(* IEC 61131-3 sources: wago_2pump_ebm_fans/PFC200_G2_2ETH_RS_CAN_DPS_T.device.xml.v3^/Plc Logic.plclogic.xml.v3^/Application.application.xml.v3^, 5 files *)

(* ---- GVL.gvl ---- *)
{attribute 'qualified_only'}
VAR_GLOBAL
	Baths: ARRAY[0..1] OF Bath;
	fan_password :STRING(6) := 'epM EC';

	QFUndervoltage:	BOOL;
	ContainerAirTemp: REAL;
	ContainerAirHumi: REAL;
	CabinetAirTemp: REAL;
	CabinetAirHumi: REAL;

	EMERGENCY:              BOOL;
END_VAR

(* ---- MODBUS.gvl ---- *)
{attribute 'qualified_only'}
VAR_GLOBAL

END_VAR

(* ---- DATA_EXTRACTOR.prg.st ---- *)
PROGRAM DATA_EXTRACTOR
VAR
	LeftIncomingTemp: INT;
	LeftOungoingTemp: INT;
	RightIncomingTemp: INT;
	RightOutgoingTemp: INT;

	LeftPressureIn: WORD;
	LeftPressureOut: WORD;
	RightPressureIn: WORD;
	RightPressureOut: WORD;

	ContainerAirTemp: WORD;
	ContainerAirHumi: WORD;

	CabinetAirTemp: WORD;
	CabinetAirHumi: WORD;

	AirTempSensorMin: REAL:= -40;
	AirTempSensorDeltaT: REAL:= 100;

	TempSensorMin: REAL:= -40;
	TempSensorDeltaT: REAL:= 100;
END_VAR;

GVL.Baths[0].LiquidInTemp := INT_TO_REAL(LeftIncomingTemp)/10;
GVL.Baths[0].LiquidOutTemp := INT_TO_REAL(LeftOungoingTemp)/10;
GVL.Baths[1].LiquidInTemp := INT_TO_REAL(RightIncomingTemp)/10;
GVL.Baths[1].LiquidOutTemp := INT_TO_REAL(RightOutgoingTemp)/10;

GVL.Baths[0].PressureIncoming := (WORD_TO_REAL(LeftPressureIn)/2047.5)/16*GVL.Baths[0].BathConfig.CalibrateInPressureSensorDelta-ABS(GVL.Baths[0].BathConfig.CalibrateInPressureSensorMIN);
GVL.Baths[0].PressureOutgoing := (WORD_TO_REAL(LeftPressureOut)/2047.5)/16*GVL.Baths[0].BathConfig.CalibrateOutPressureSensorDelta-ABS(GVL.Baths[0].BathConfig.CalibrateOutPressureSensorMIN);
GVL.Baths[1].PressureIncoming := (WORD_TO_REAL(RightPressureIn)/2047.5)/16*GVL.Baths[1].BathConfig.CalibrateInPressureSensorDelta-ABS(GVL.Baths[1].BathConfig.CalibrateInPressureSensorMIN);
GVL.Baths[1].PressureOutgoing := (WORD_TO_REAL(RightPressureOut)/2047.5)/16*GVL.Baths[1].BathConfig.CalibrateOutPressureSensorDelta-ABS(GVL.Baths[1].BathConfig.CalibrateOutPressureSensorMIN);

GVL.Baths[0].PressureIncomingBar := GVL.Baths[0].PressureIncoming/14.5038;
GVL.Baths[0].PressureOutgoingBar := GVL.Baths[0].PressureOutgoing/14.5038;
GVL.Baths[1].PressureIncomingBar := GVL.Baths[1].PressureIncoming/14.5038;
GVL.Baths[1].PressureOutgoingBar := GVL.Baths[1].PressureOutgoing/14.5038;

GVL.ContainerAirTemp:= (WORD_TO_REAL(ContainerAirTemp)/2047.5)/16*AirTempSensorDeltaT-ABS(AirTempSensorMin);
GVL.ContainerAirHumi := (WORD_TO_REAL(CabinetAirHumi)/2047.5)/16*100;

GVL.CabinetAirTemp:= (WORD_TO_REAL(CabinetAirTemp)/2047.5)/16*AirTempSensorDeltaT-ABS(AirTempSensorMin);
GVL.CabinetAirHumi := (WORD_TO_REAL(CabinetAirHumi)/2047.5)/16*100;

(* ---- PLC_PRG.prg.st ---- *)
PROGRAM PLC_PRG
VAR
	START 	:BOOL;
END_VAR;

START := TRUE;

(* ---- TIMERS.prg.st ---- *)
PROGRAM TIMERS
VAR
	QF1_ENABLE_TOF : TOF;
	QF1_DISABLE_TOF : TOF;

	QF2_ENABLE_TOF : TOF;
	QF2_DISABLE_TOF : TOF;
END_VAR;

(* Enabling QF1 *)
IF GVL.Baths[0].MainRelayDisable = FALSE THEN
	IF GVL.Baths[0].MainRelayEnable = TRUE THEN
		GVL.Baths[0].MainRelay_on := FALSE;
		GVL.Baths[0].MainRelayStatus := TRUE;
	END_IF;
	QF1_ENABLE_TOF(IN := GVL.Baths[0].MainRelay_on, PT := T#2S);
	GVL.Baths[0].MainRelayEnable := QF1_ENABLE_TOF.Q;
END_IF

IF GVL.Baths[0].MainRelayEnable = FALSE THEN
	IF GVL.Baths[0].MainRelayDisable = TRUE THEN
		GVL.Baths[0].MainRelay_off := FALSE;
		GVL.Baths[0].MainRelayStatus := FALSE;
	END_IF;
	QF1_DISABLE_TOF(IN := GVL.Baths[0].MainRelay_off, PT := T#5S);
	GVL.Baths[0].MainRelayDisable := QF1_DISABLE_TOF.Q;
END_IF;

(* Enabling QF2 *)
IF GVL.Baths[1].MainRelayDisable = FALSE THEN
	IF GVL.Baths[1].MainRelayEnable = TRUE THEN
		GVL.Baths[1].MainRelay_on := FALSE;
		GVL.Baths[1].MainRelayStatus := TRUE;
	END_IF;
	QF2_ENABLE_TOF(IN := GVL.Baths[1].MainRelay_on, PT := T#2S);
	GVL.Baths[1].MainRelayEnable := QF2_ENABLE_TOF.Q;
END_IF

(* Enabling QF2 *)
IF GVL.Baths[1].MainRelayEnable = FALSE THEN
	IF GVL.Baths[1].MainRelayDisable = TRUE THEN
		GVL.Baths[1].MainRelay_off := FALSE;
		GVL.Baths[1].MainRelayStatus := FALSE;
	END_IF;
	QF2_DISABLE_TOF(IN := GVL.Baths[1].MainRelay_off, PT := T#5S);
	GVL.Baths[1].MainRelayDisable := QF2_DISABLE_TOF.Q;
END_IF;

IF GVL.Baths[0].BathConfig.AdminFanRelay = ENUM_AdminRelayStatus.relayForceEnable THEN
	GVL.Baths[0].MainKMStatus := TRUE;
END_IF;

IF GVL.Baths[0].BathConfig.AdminFanRelay = ENUM_AdminRelayStatus.relayForceDisable THEN
	GVL.Baths[0].MainKMStatus := FALSE;
END_IF;

IF GVL.Baths[1].BathConfig.AdminFanRelay = ENUM_AdminRelayStatus.relayForceEnable THEN
	GVL.Baths[1].MainKMStatus := TRUE;
END_IF;

IF GVL.Baths[1].BathConfig.AdminFanRelay = ENUM_AdminRelayStatus.relayForceDisable THEN
	GVL.Baths[1].MainKMStatus := FALSE;
END_IF;

IF GVL.Baths[0].BathConfig.AdminPumpRelay = ENUM_AdminRelayStatus.relayForceEnable THEN
	GVL.Baths[0].PumpKMStatus := TRUE;
END_IF;

IF GVL.Baths[0].BathConfig.AdminPumpRelay = ENUM_AdminRelayStatus.relayForceDisable THEN
	GVL.Baths[0].PumpKMStatus := FALSE;
END_IF;

IF GVL.Baths[1].BathConfig.AdminPumpRelay = ENUM_AdminRelayStatus.relayForceEnable THEN
	GVL.Baths[1].PumpKMStatus := TRUE;
END_IF

IF GVL.Baths[1].BathConfig.AdminPumpRelay = ENUM_AdminRelayStatus.relayForceDisable THEN
	GVL.Baths[1].PumpKMStatus := FALSE;
END_IF
